FUNCTION_BLOCK SelectAutoValue (* Basic Function Block Type *)
  (* Standard: 61499-2 *)
  (* Version 0.0, 2011-12-29, 4DIAC-IDE, 4DIAC-Consortium *)
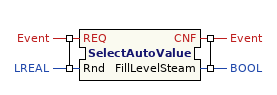
  EVENT_INPUT
    REQ WITH Rnd; (* Normal Execution Request *)
  END_EVENT
  EVENT_OUTPUT
    CNF WITH FillLevelSteam; (* Execution Confirmation *)
  END_EVENT
  VAR_INPUT
    Rnd : LREAL; (* Input event qualifier *)
  END_VAR
  VAR_OUTPUT
    FillLevelSteam : BOOL; (* Output event qualifier *)
  END_VAR
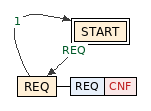
  EC_STATES
    START; (* Initial State *)
    REQ : REQ -> CNF; (* Normal execution *)
  END_STATES
  EC_TRANSITIONS
    START TO REQ := REQ;
    REQ TO START := 1;
  END_TRANSITIONS
  ALGORITHM REQ IN ST: (* Normally executed algorithm *)
IF Rnd > 1.0 THEN
	FillLevelSteam:=1;
ELSE
		FillLevelSteam:=0;
END_IF;
  END_ALGORITHM
END_FUNCTION_BLOCK
